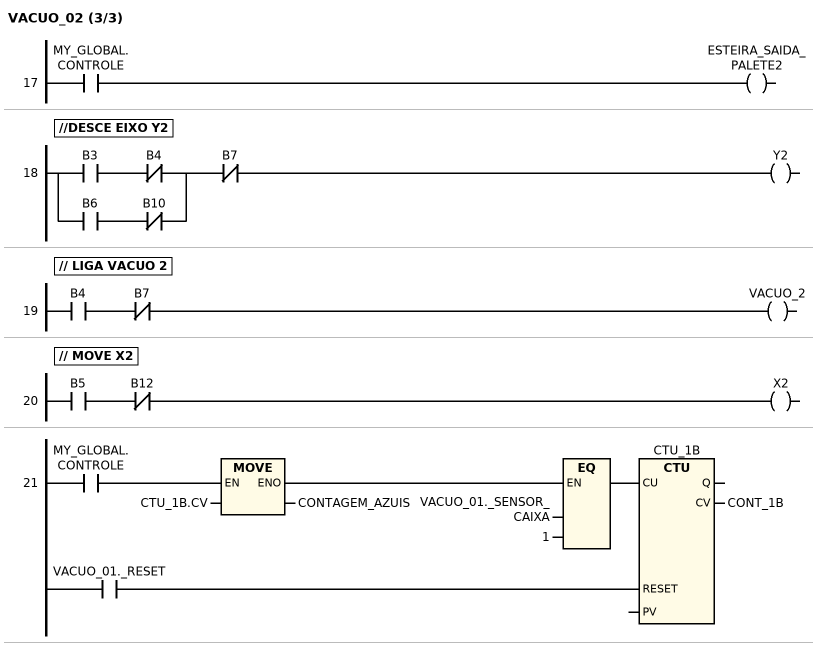
// NETWORK 17
ESTEIRA_SAIDA_PALETE2 := MY_GLOBAL.CONTROLE;

// NETWORK 18
// label: //DESCE EIXO Y2
Y2 := (B3 AND NOT B4 OR B6 AND NOT B10) AND NOT B7;

// NETWORK 19
// label: // LIGA VACUO 2
VACUO_2 := B4 AND NOT B7;

// NETWORK 20
// label: // MOVE X2
X2 := B5 AND NOT B12;

// NETWORK 21
_w4 := MY_GLOBAL.CONTROLE;
IF _w4 THEN CONTAGEM_AZUIS := CTU_1B.CV; END_IF
CTU_1B(CU := _w4 AND VACUO_01._SENSOR_CAIXA = 1, RESET := VACUO_01._RESET, CV => CONT_1B); // CTU

END_PROGRAM

// Device/Application/PALETIZADOR_01
PROGRAM PALETIZADOR_01
VAR
//PALLETIZADOR N01 (PARTE DE CIMA)
	//ENTRADAS
	_SENSOR_ENTRADA_CAIXA1:BOOL; // CONTA AS CAIXAS QUE VÃO PARA O PALLET CENTRALIZADOR1:BOOL;
	
	//SAIDAS
	EMPURRADOR1:BOOL;
	CENTRALIZADOR1:BOOL;
	PLACA1:BOOL;
	ESTEIRA_PALETIZADOR1:BOOL;
	ESTEIRA_SECUNDARIA1_1:BOOL;
	
// PALETIZADOR N01 (PARTE DO MEIO)
	//SAIDAS
	MOVER1:BOOL;
	DESCER1:BOOL;
	SUBIR1:BOOL; 
	
// PALETIZADOR N01 (PARTE DE BAIXO)
	//ENTRADAS
	_SENSOR_P1:BOOL;
	
	//SAIDAS
	ESTEIRA_ELEVADOR1:BOOL;
	ESTEIRA_PALETE1:BOOL;
	
// AUXILIARES
    C1:BOOL;  // AUXILIA NO ACIONAMENTO DO TEMPORIZADOR QUE ACIONA O EMPURRADOR 1
    C2:BOOL;  // AUXILIA NO ACIONAMENTO DO TEMPORIZADOR QUE ACIONA O CENTRALIZADOR 1
    C3:BOOL;  // AUXILIA NO ACIONAMENTO DO TEMPORIZADOR QUE ACIONA A PORTA 1 
    C4:BOOL;  // AUXILIA NO ACIONAMENTO DO TEMPORIZADOR QUE DESACIONA O EMPURRADOR 1 E O CENTRALIZADOR 1
    C5:BOOL;  // AUXILIA NO ACIONAMENTO DO TEMPORIZADOR QUE DESACIONA A PORTA 1 
    C6:BOOL;  // AUXILIA NO ACIONAMENTO DO RESET DO CONTADOR DE CAIXAS VERDES 
    C7:BOOL;  // AUXILIA NO ACIONAMENTO DO TEMPORIZADOR QUE CONTA O TEMPO DE ESPERA PARA O ELEVADOR DO PALET 1 DESCER    
	C8:BOOL;  // AUXILIA NO ACIONMENTO DO TEMPORIZADOR QUE CONTA O TEMPO DE DESCIDA DO ELEVADOR DO PALET 1
	C9:BOOL;  // AUXILIA PERMITINDO A SUBIDA DO ELEVADOR DO PALET 1 DEPOIS DO CONTADOR CONTAR DUAS CAIXAS VERDES 
	C10:BOOL;  // AUXILIA NO ACIONAMENTO DA ESTEIRA DO ELEVADOR E DA ESTEIRA DO PALET 1 COM O PALET E AS CAIXAS  
	C11:BOOL;  // AUXILIA NO ACIONAMENTO DO TEMPORIZADOR QUE CONTA O TEMPO DE SAIDA DO PALET COM A CAIXA DO PALETIZADOR 1 
	C12:BOOL;  // AUXILIA NA PARTE FINAL DO PROCESSO 
	C13:BOOL;  // AUXILIA IMPEDINDO O ACIONAMENTO DA ESTEIRA DAS CAIXAS VERDES E DA ESTEIRA DE CIMA DO PALET 1 ENQUANDO O ELEVADOR DO PALET 1 ESTÁ ACIONADO  
	
// TEMPORIZADORES
    TON_1C: TON;
	TEMPO_1C: TIME;
	TON_2C: TON;
	TEMPO_2C: TIME;
	TON_3C: TON;
	TEMPO_3C: TIME;
	TON_4C: TON;
	TEMPO_4C: TIME;
	TON_5C: TON;
	TEMPO_5C: TIME;
	TON_6C: TON;
	TEMPO_6C: TIME;
	TON_7C: TON;
	TEMPO_7C: TIME;
	TON_8C: TON;
	TEMPO_8C: TIME;
	TON_9C: TON;
	TEMPO_9C: TIME;
	
// CONTADORES 
	CTU_1C: CTU;
	CONT_1C: WORD;

END_VAR
VAR // added by the converter: edge detectors and wires of the graphical bodies
    _w1, _w2 : BOOL;
END_VAR

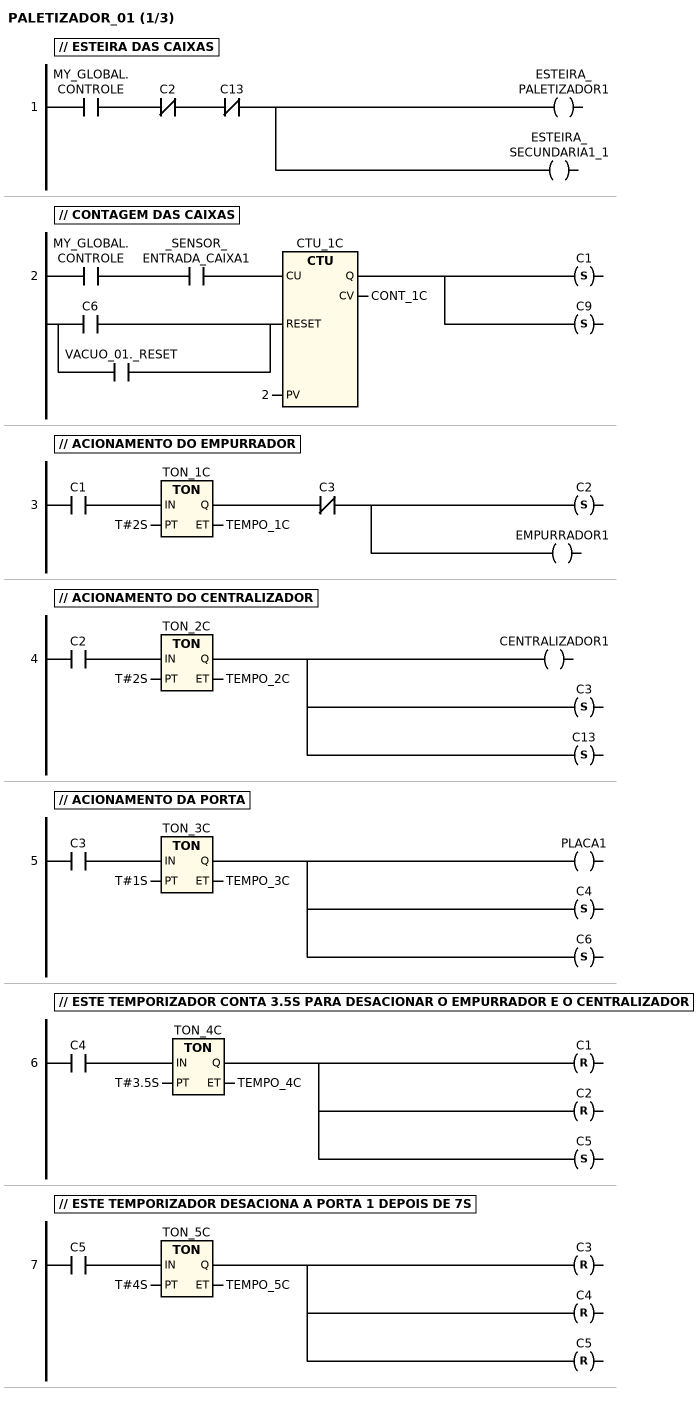
// NETWORK 1
// label: // ESTEIRA DAS CAIXAS
_w1 := MY_GLOBAL.CONTROLE AND NOT C2 AND NOT C13;
ESTEIRA_PALETIZADOR1 := _w1;
ESTEIRA_SECUNDARIA1_1 := _w1;

// NETWORK 2
// label: // CONTAGEM DAS CAIXAS
CTU_1C(
    CU := MY_GLOBAL.CONTROLE AND _SENSOR_ENTRADA_CAIXA1,
    RESET := C6 OR VACUO_01._RESET,
    PV := 2,
    CV => CONT_1C); // CTU
C1 S= CTU_1C.Q;
C9 S= CTU_1C.Q;

// NETWORK 3
// label: // ACIONAMENTO DO EMPURRADOR
TON_1C(IN := C1, PT := T#2S, ET => TEMPO_1C); // TON
_w2 := TON_1C.Q AND NOT C3;
C2 S= _w2;
EMPURRADOR1 := _w2;

// NETWORK 4
// label: // ACIONAMENTO DO CENTRALIZADOR
TON_2C(IN := C2, PT := T#2S, ET => TEMPO_2C); // TON
CENTRALIZADOR1 := TON_2C.Q;
C3 S= TON_2C.Q;
C13 S= TON_2C.Q;

// NETWORK 5
// label: // ACIONAMENTO DA PORTA
TON_3C(IN := C3, PT := T#1S, ET => TEMPO_3C); // TON
PLACA1 := TON_3C.Q;
C4 S= TON_3C.Q;
C6 S= TON_3C.Q;

// NETWORK 6
// label: // ESTE TEMPORIZADOR CONTA 3.5S PARA DESACIONAR O EMPURRADOR E O CENTRALIZADOR
TON_4C(IN := C4, PT := T#3.5S, ET => TEMPO_4C); // TON
C1 R= TON_4C.Q;
C2 R= TON_4C.Q;
C5 S= TON_4C.Q;

// NETWORK 7
// label: // ESTE TEMPORIZADOR DESACIONA A PORTA 1 DEPOIS DE 7S
TON_5C(IN := C5, PT := T#4S, ET => TEMPO_5C); // TON
C3 R= TON_5C.Q;
C4 R= TON_5C.Q;
C5 R= TON_5C.Q;

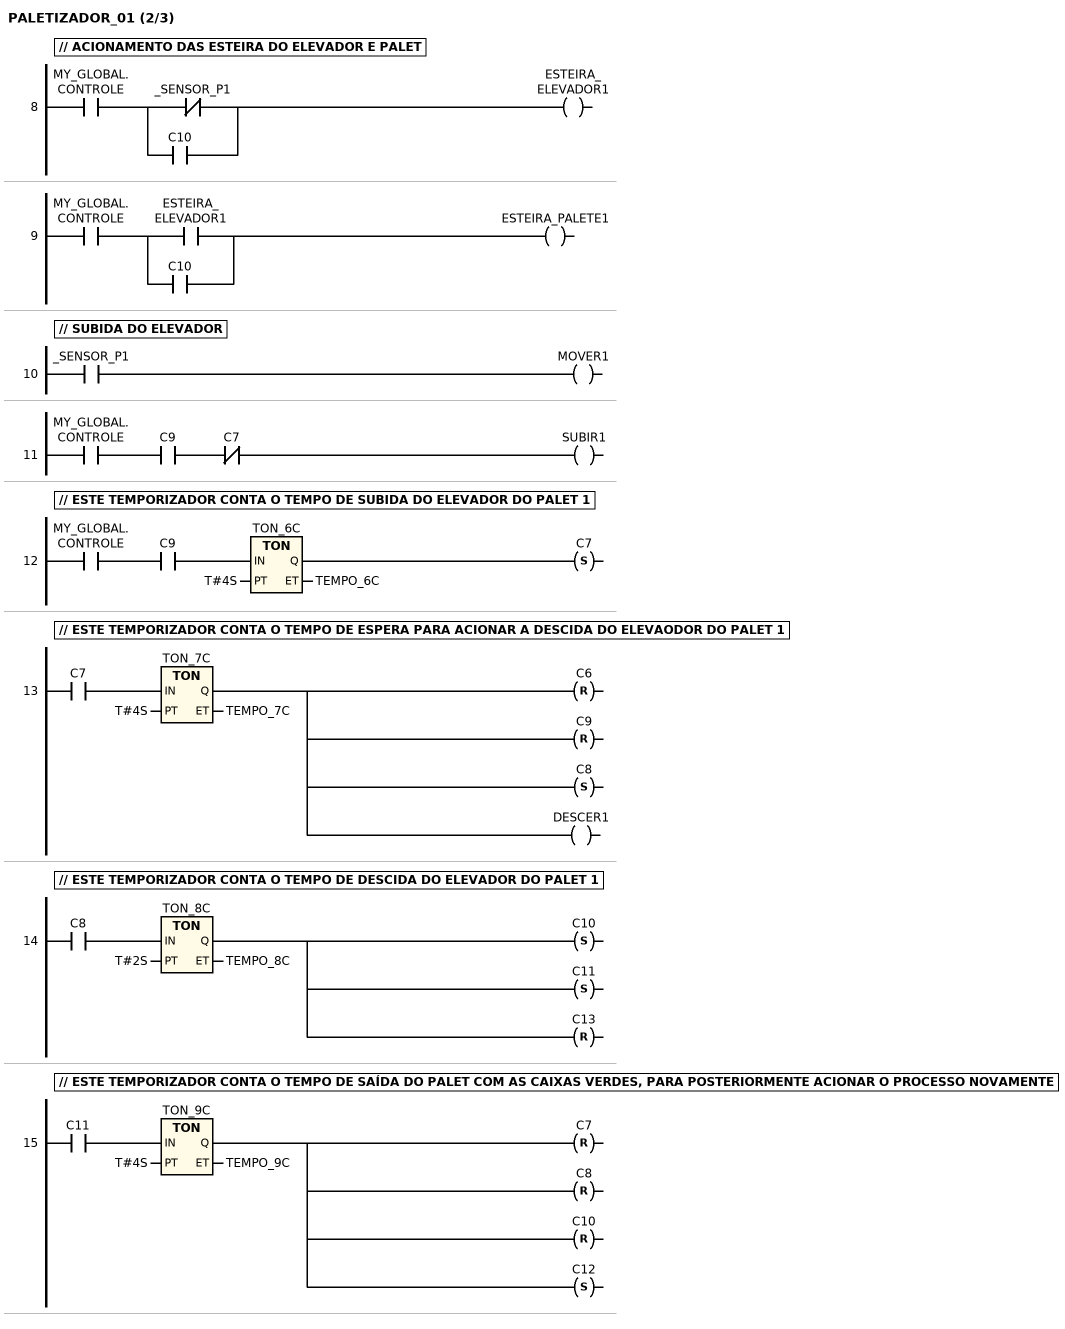
// NETWORK 8
// label: // ACIONAMENTO DAS ESTEIRA DO ELEVADOR E PALET
ESTEIRA_ELEVADOR1 := MY_GLOBAL.CONTROLE AND (NOT _SENSOR_P1 OR C10);

// NETWORK 9
ESTEIRA_PALETE1 := MY_GLOBAL.CONTROLE AND (ESTEIRA_ELEVADOR1 OR C10);

// NETWORK 10
// label: // SUBIDA DO ELEVADOR
MOVER1 := _SENSOR_P1;

// NETWORK 11
SUBIR1 := MY_GLOBAL.CONTROLE AND C9 AND NOT C7;

// NETWORK 12
// label: // ESTE TEMPORIZADOR CONTA O TEMPO DE SUBIDA DO ELEVADOR DO PALET 1
TON_6C(IN := MY_GLOBAL.CONTROLE AND C9, PT := T#4S, ET => TEMPO_6C); // TON
C7 S= TON_6C.Q;

// NETWORK 13
// label: // ESTE TEMPORIZADOR CONTA O TEMPO DE ESPERA PARA ACIONAR A DESCIDA DO ELEVAODOR DO PALET 1
TON_7C(IN := C7, PT := T#4S, ET => TEMPO_7C); // TON
C6 R= TON_7C.Q;
C9 R= TON_7C.Q;
C8 S= TON_7C.Q;
DESCER1 := TON_7C.Q;

// NETWORK 14
// label: // ESTE TEMPORIZADOR CONTA O TEMPO DE DESCIDA DO ELEVADOR DO PALET 1
TON_8C(IN := C8, PT := T#2S, ET => TEMPO_8C); // TON
C10 S= TON_8C.Q;
C11 S= TON_8C.Q;
C13 R= TON_8C.Q;

// NETWORK 15
// label: // ESTE TEMPORIZADOR CONTA O TEMPO DE SAÍDA DO PALET COM AS CAIXAS VERDES, PARA POSTERIORMENTE ACIONAR O PROCESSO NOVAMENTE
TON_9C(IN := C11, PT := T#4S, ET => TEMPO_9C); // TON
C7 R= TON_9C.Q;
C8 R= TON_9C.Q;
C10 R= TON_9C.Q;
C12 S= TON_9C.Q;

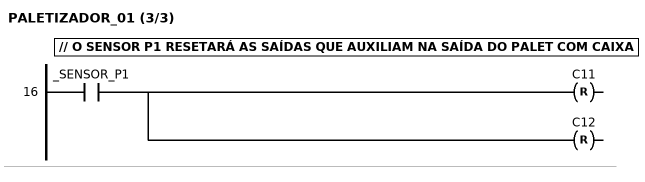
// NETWORK 16
// label: // O SENSOR P1 RESETARÁ AS SAÍDAS QUE AUXILIAM NA SAÍDA DO PALET COM CAIXA
C11 R= _SENSOR_P1;
C12 R= _SENSOR_P1;

END_PROGRAM

// Device/Application/PALETIZADOR_02
PROGRAM PALETIZADOR_02
VAR
//PALLETIZADOR N02 (PARTE DE CIMA)
	//ENTRADAS
	_SENSOR_ENTRADA_CAIXA2:BOOL; // CONTA AS CAIXAS QUE VÃO PARA O PALLET CENTRALIZADOR1:BOOL;
	
	//SAIDAS
	EMPURRADOR2:BOOL;
	CENTRALIZADOR2:BOOL;
	PLACA2:BOOL;
	ESTEIRA_PALETIZADOR2:BOOL;
	ESTEIRA_SECUNDARIA2_1:BOOL;
	
// PALETIZADOR N02 (PARTE DO MEIO)
	//SAIDAS
	MOVER2:BOOL;
	DESCER2:BOOL;
	SUBIR2:BOOL; 
	
// PALETIZADOR N02 (PARTE DE BAIXO)
	//ENTRADAS
	_SENSOR_P2:BOOL;
	
	//SAIDAS
	ESTEIRA_ELEVADOR2:BOOL;
	ESTEIRA_PALETE2:BOOL;
	
// AUXILIARES
    D1:BOOL;  // AUXILIA NO ACIONAMENTO DO TEMPORIZADOR QUE ACIONA O EMPURRADOR 1
    D2:BOOL;  // AUXILIA NO ACIONAMENTO DO TEMPORIZADOR QUE ACIONA O CENTRALIZADOR 1
    D3:BOOL;  // AUXILIA NO ACIONAMENTO DO TEMPORIZADOR QUE ACIONA A PORTA 1 
    D4:BOOL;  // AUXILIA NO ACIONAMENTO DO TEMPORIZADOR QUE DESACIONA O EMPURRADOR 1 E O CENTRALIZADOR 1
    D5:BOOL;  // AUXILIA NO ACIONAMENTO DO TEMPORIZADOR QUE DESACIONA A PORTA 1 
    D6:BOOL;  // AUXILIA NO ACIONAMENTO DO RESET DO CONTADOR DE CAIXAS VERDES 
    D7:BOOL;  // AUXILIA NO ACIONAMENTO DO TEMPORIZADOR QUE CONTA O TEMPO DE ESPERA PARA O ELEVADOR DO PALET 1 DESCER    
	D8:BOOL;  // AUXILIA NO ACIONMENTO DO TEMPORIZADOR QUE CONTA O TEMPO DE DESCIDA DO ELEVADOR DO PALET 1
	D9:BOOL;  // AUXILIA PERMITINDO A SUBIDA DO ELEVADOR DO PALET 1 DEPOIS DO CONTADOR CONTAR DUAS CAIXAS VERDES 
	D10:BOOL;  // AUXILIA NO ACIONAMENTO DA ESTEIRA DO ELEVADOR E DA ESTEIRA DO PALET 1 COM O PALET E AS CAIXAS  
	D11:BOOL;  // AUXILIA NO ACIONAMENTO DO TEMPORIZADOR QUE CONTA O TEMPO DE SAIDA DO PALET COM A CAIXA DO PALETIZADOR 1 
	D12:BOOL;  // AUXILIA NA PARTE FINAL DO PROCESSO 
	D13:BOOL;  // AUXILIA IMPEDINDO O ACIONAMENTO DA ESTEIRA DAS CAIXAS VERDES E DA ESTEIRA DE CIMA DO PALET 1 ENQUANDO O ELEVADOR DO PALET 1 ESTÁ ACIONADO  
	
// TEMPORIZADORES
    TON_1D: TON;
	TEMPO_1D: TIME;
	TON_2D: TON;
	TEMPO_2D: TIME;
	TON_3D: TON;
	TEMPO_3D: TIME;
	TON_4D: TON;
	TEMPO_4D: TIME;
	TON_5D: TON;
	TEMPO_5D: TIME;
	TON_6D: TON;
	TEMPO_6D: TIME;
	TON_7D: TON;
	TEMPO_7D: TIME;
	TON_8D: TON;
	TEMPO_8D: TIME;
	TON_9D: TON;
	TEMPO_9D: TIME;
	
// CONTADORES 
	CTU_1D: CTU;
	CONT_1D: WORD;

END_VAR
VAR // added by the converter: edge detectors and wires of the graphical bodies
    _w1, _w2 : BOOL;
END_VAR

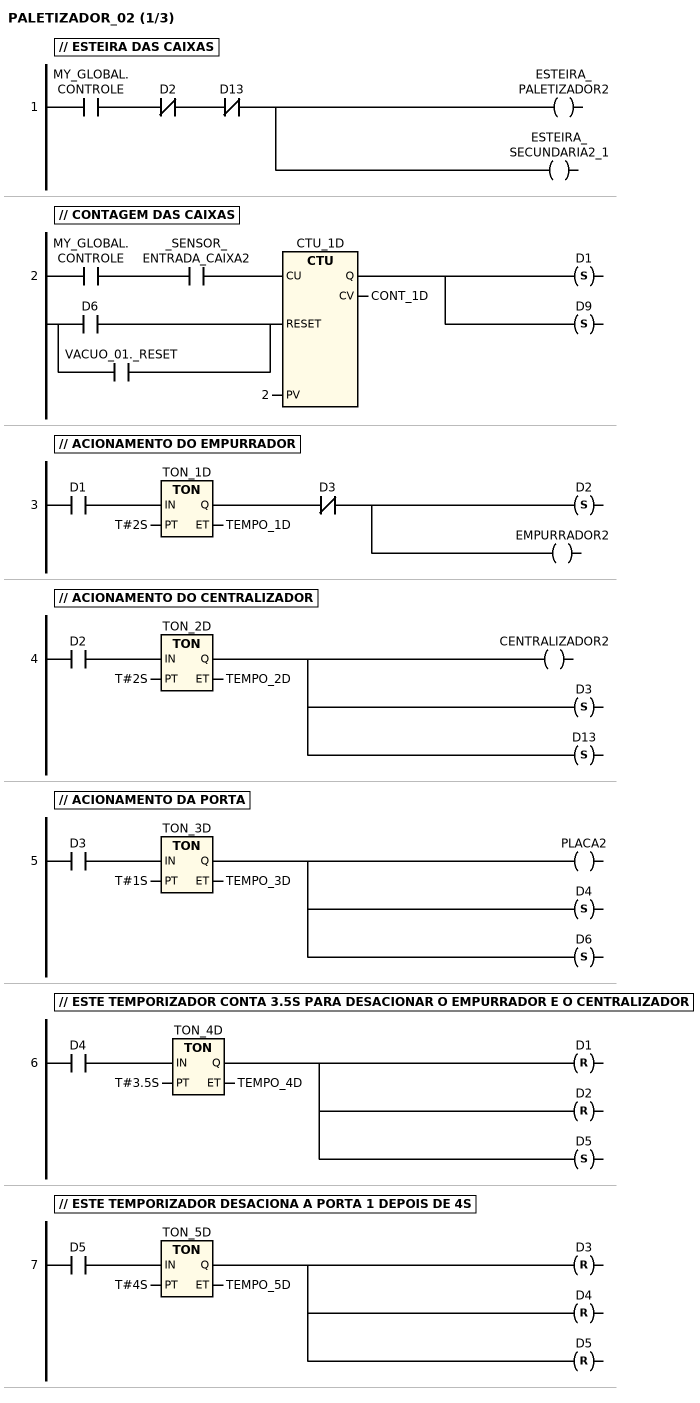
// NETWORK 1
// label: // ESTEIRA DAS CAIXAS
_w1 := MY_GLOBAL.CONTROLE AND NOT D2 AND NOT D13;
ESTEIRA_PALETIZADOR2 := _w1;
ESTEIRA_SECUNDARIA2_1 := _w1;

// NETWORK 2
// label: // CONTAGEM DAS CAIXAS
CTU_1D(
    CU := MY_GLOBAL.CONTROLE AND _SENSOR_ENTRADA_CAIXA2,
    RESET := D6 OR VACUO_01._RESET,
    PV := 2,
    CV => CONT_1D); // CTU
D1 S= CTU_1D.Q;
D9 S= CTU_1D.Q;

// NETWORK 3
// label: // ACIONAMENTO DO EMPURRADOR
TON_1D(IN := D1, PT := T#2S, ET => TEMPO_1D); // TON
_w2 := TON_1D.Q AND NOT D3;
D2 S= _w2;
EMPURRADOR2 := _w2;

// NETWORK 4
// label: // ACIONAMENTO DO CENTRALIZADOR
TON_2D(IN := D2, PT := T#2S, ET => TEMPO_2D); // TON
CENTRALIZADOR2 := TON_2D.Q;
D3 S= TON_2D.Q;
D13 S= TON_2D.Q;

// NETWORK 5
// label: // ACIONAMENTO DA PORTA
TON_3D(IN := D3, PT := T#1S, ET => TEMPO_3D); // TON
PLACA2 := TON_3D.Q;
D4 S= TON_3D.Q;
D6 S= TON_3D.Q;

// NETWORK 6
// label: // ESTE TEMPORIZADOR CONTA 3.5S PARA DESACIONAR O EMPURRADOR E O CENTRALIZADOR
TON_4D(IN := D4, PT := T#3.5S, ET => TEMPO_4D); // TON
D1 R= TON_4D.Q;
D2 R= TON_4D.Q;
D5 S= TON_4D.Q;

// NETWORK 7
// label: // ESTE TEMPORIZADOR DESACIONA A PORTA 1 DEPOIS DE 4S
TON_5D(IN := D5, PT := T#4S, ET => TEMPO_5D); // TON
D3 R= TON_5D.Q;
D4 R= TON_5D.Q;
D5 R= TON_5D.Q;

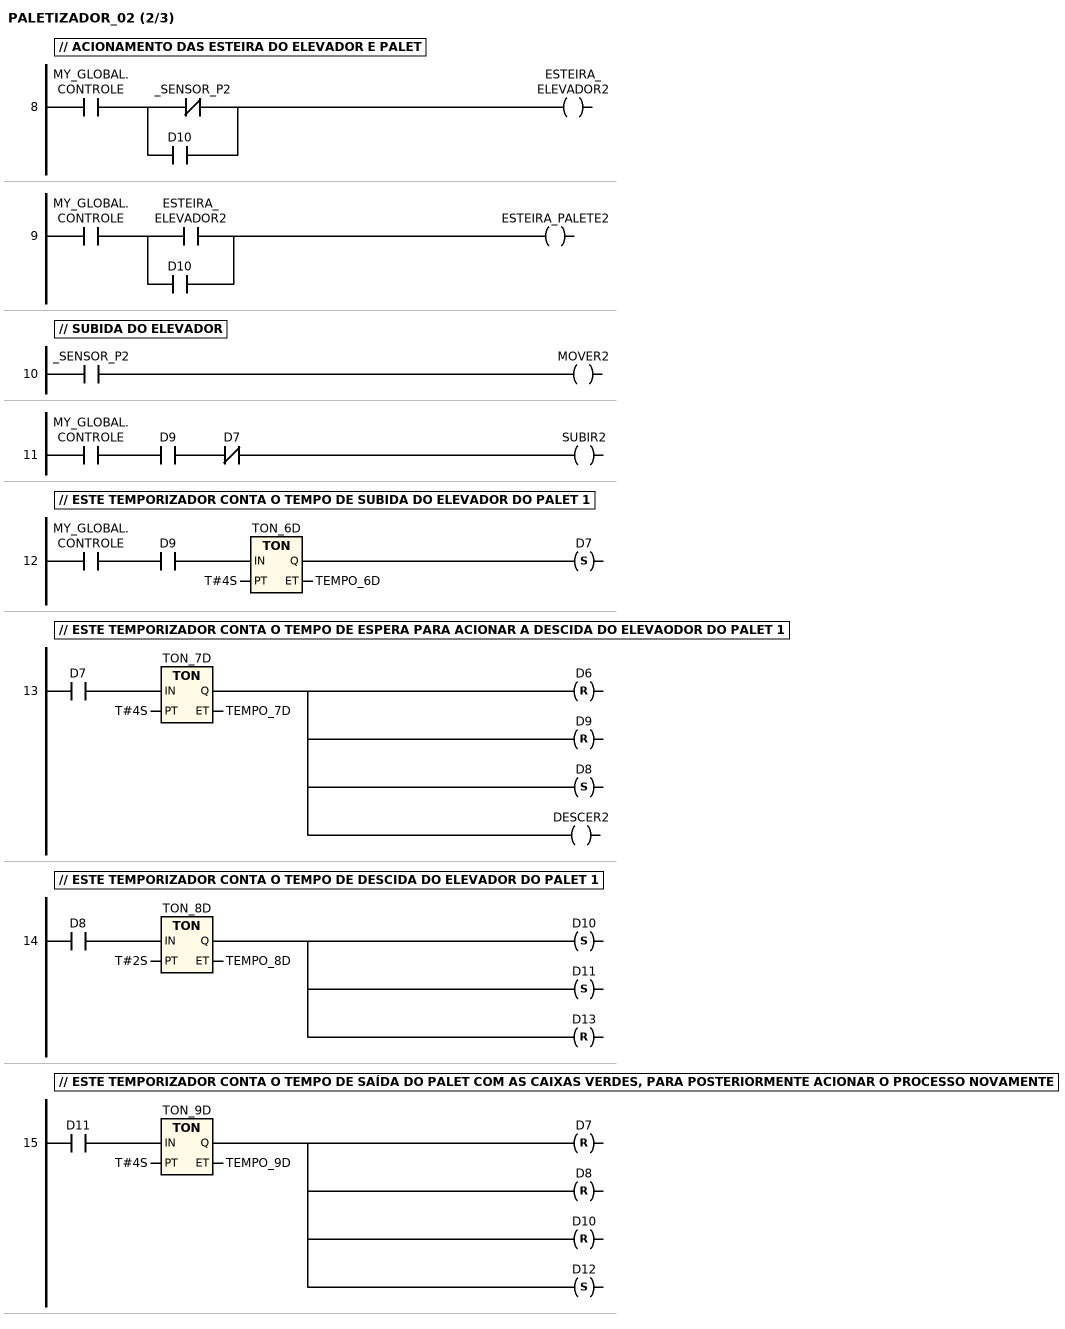
// NETWORK 8
// label: // ACIONAMENTO DAS ESTEIRA DO ELEVADOR E PALET
ESTEIRA_ELEVADOR2 := MY_GLOBAL.CONTROLE AND (NOT _SENSOR_P2 OR D10);

// NETWORK 9
ESTEIRA_PALETE2 := MY_GLOBAL.CONTROLE AND (ESTEIRA_ELEVADOR2 OR D10);

// NETWORK 10
// label: // SUBIDA DO ELEVADOR
MOVER2 := _SENSOR_P2;

// NETWORK 11
SUBIR2 := MY_GLOBAL.CONTROLE AND D9 AND NOT D7;

// NETWORK 12
// label: // ESTE TEMPORIZADOR CONTA O TEMPO DE SUBIDA DO ELEVADOR DO PALET 1
TON_6D(IN := MY_GLOBAL.CONTROLE AND D9, PT := T#4S, ET => TEMPO_6D); // TON
D7 S= TON_6D.Q;

// NETWORK 13
// label: // ESTE TEMPORIZADOR CONTA O TEMPO DE ESPERA PARA ACIONAR A DESCIDA DO ELEVAODOR DO PALET 1
TON_7D(IN := D7, PT := T#4S, ET => TEMPO_7D); // TON
D6 R= TON_7D.Q;
D9 R= TON_7D.Q;
D8 S= TON_7D.Q;
DESCER2 := TON_7D.Q;

// NETWORK 14
// label: // ESTE TEMPORIZADOR CONTA O TEMPO DE DESCIDA DO ELEVADOR DO PALET 1
TON_8D(IN := D8, PT := T#2S, ET => TEMPO_8D); // TON
D10 S= TON_8D.Q;
D11 S= TON_8D.Q;
D13 R= TON_8D.Q;

// NETWORK 15
// label: // ESTE TEMPORIZADOR CONTA O TEMPO DE SAÍDA DO PALET COM AS CAIXAS VERDES, PARA POSTERIORMENTE ACIONAR O PROCESSO NOVAMENTE
TON_9D(IN := D11, PT := T#4S, ET => TEMPO_9D); // TON
D7 R= TON_9D.Q;
D8 R= TON_9D.Q;
D10 R= TON_9D.Q;
D12 S= TON_9D.Q;

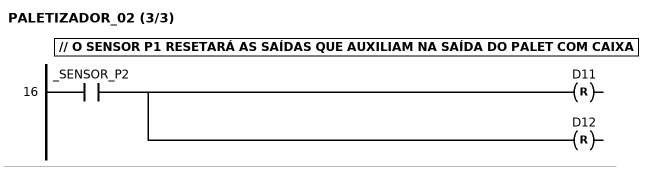
// NETWORK 16
// label: // O SENSOR P1 RESETARÁ AS SAÍDAS QUE AUXILIAM NA SAÍDA DO PALET COM CAIXA
D11 R= _SENSOR_P2;
D12 R= _SENSOR_P2;

END_PROGRAM
